FUNCTION_BLOCK FB_System_HES_991
VAR_INPUT
	Freigabe_auto				: BOOL;
	Freigabe_Deakt_auto			: BOOL;
	Betrieb_Anford_auto			: BOOL;

END_VAR
VAR_OUTPUT
	{attribute 'OPC.UA.DA' := '1'}Steuerung				: ST_System_HES_Steuerung;		
	{attribute 'OPC.UA.DA' := '1'}Stellwert				: ST_System_HES_Stellwert;		
	{attribute 'OPC.UA.DA' := '1'}Zustand					: ST_System_HES_Zustand;	
	{attribute 'OPC.UA.DA' := '1'}Parameter				: ST_System_HES_Parameter;		
END_VAR
VAR
	Pumpe_191					: FB_PU_191;
	Stellventil_191				: FB_SV;
	HybriderEnergiespeicher_991	: FB_HES;

	Zustandscheck			: FB_System_HES_Zustandscheck;
	Logik					: FB_System_HES_Logik;
	Ablaufsteuerung			: FB_System_HES_Ablaufsteuerung;
	Ablaufsteuerung_191		: FB_System_HES_Ablaufsteuerung;

END_VAR
VAR // added by the converter: edge detectors and wires of the graphical bodies
    _w1, _w4, _w6 : ANY;
    _w2, _w3, _w5 : BOOL;
END_VAR

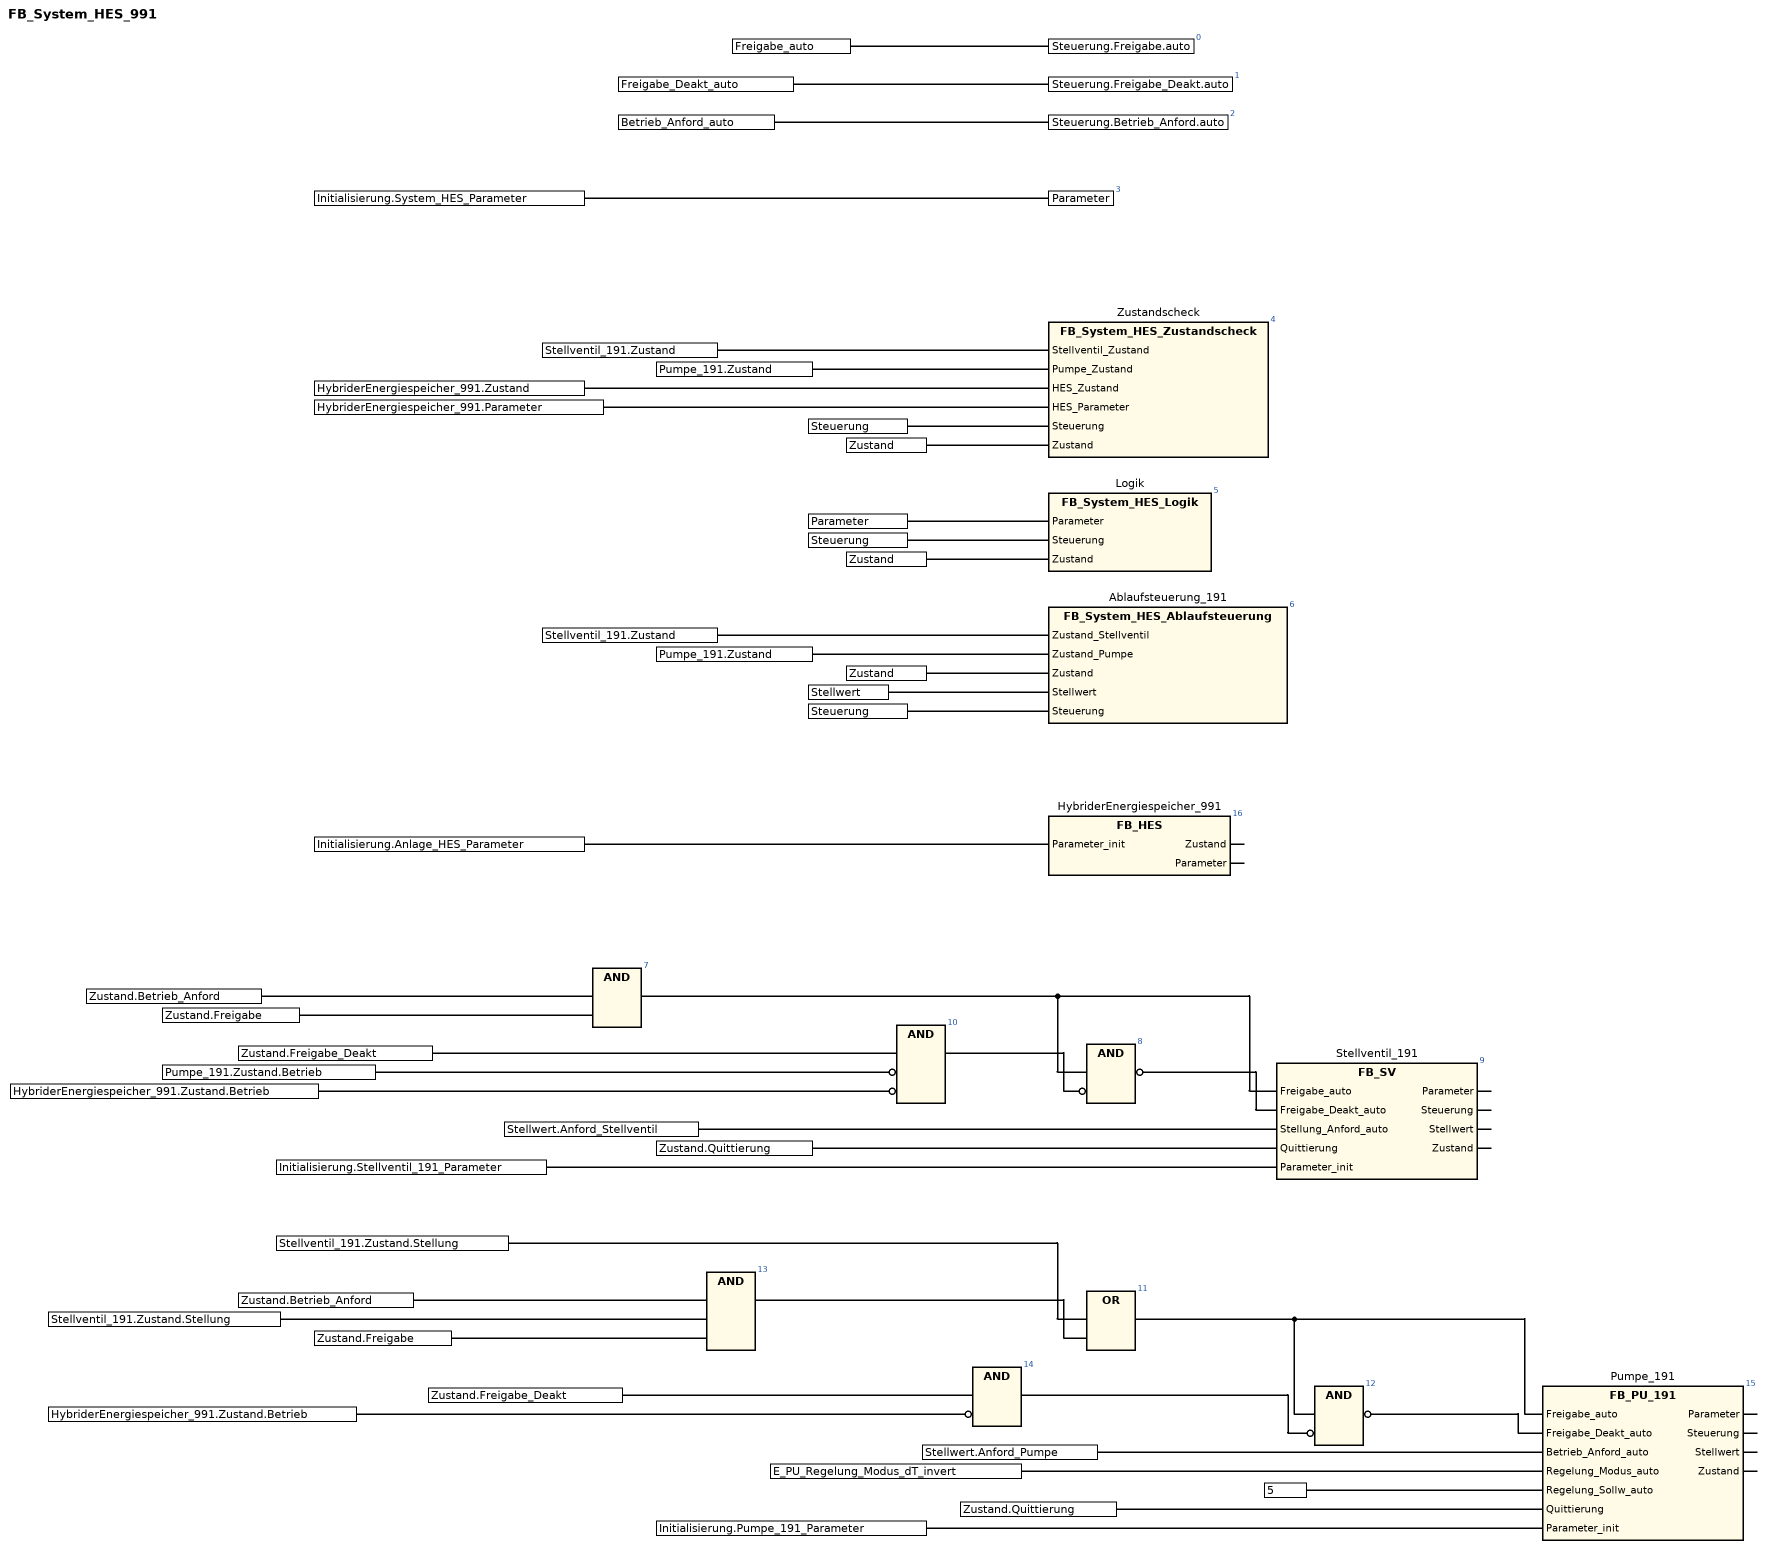
Steuerung.Freigabe.auto := Freigabe_auto;
Steuerung.Freigabe_Deakt.auto := Freigabe_Deakt_auto;
Steuerung.Betrieb_Anford.auto := Betrieb_Anford_auto;
Parameter := Initialisierung.System_HES_Parameter;
Zustandscheck(
    Stellventil_Zustand := Stellventil_191.Zustand,
    Pumpe_Zustand := Pumpe_191.Zustand,
    HES_Zustand := HybriderEnergiespeicher_991.Zustand,
    HES_Parameter := HybriderEnergiespeicher_991.Parameter,
    Steuerung := Steuerung,
    Zustand := Zustand); // FB_System_HES_Zustandscheck
Logik(Parameter := Parameter, Steuerung := Steuerung, Zustand := Zustand); // FB_System_HES_Logik
Ablaufsteuerung_191(
    Zustand_Stellventil := Stellventil_191.Zustand,
    Zustand_Pumpe := Pumpe_191.Zustand,
    Zustand := Zustand,
    Stellwert := Stellwert,
    Steuerung := Steuerung); // FB_System_HES_Ablaufsteuerung
_w1 := Zustand.Betrieb_Anford AND Zustand.Freigabe;
Stellventil_191(
    Freigabe_auto := _w1,
    Freigabe_Deakt_auto := NOT (_w1 AND NOT _w2),
    Stellung_Anford_auto := Stellwert.Anford_Stellventil,
    Quittierung := Zustand.Quittierung,
    Parameter_init := Initialisierung.Stellventil_191_Parameter); // FB_SV
_w2 := Zustand.Freigabe_Deakt AND NOT Pumpe_191.Zustand.Betrieb AND NOT HybriderEnergiespeicher_991.Zustand.Betrieb;
_w4 := Stellventil_191.Zustand.Stellung OR _w3;
_w6 := _w4 AND NOT _w5;
_w3 := Zustand.Betrieb_Anford AND Stellventil_191.Zustand.Stellung AND Zustand.Freigabe;
_w5 := Zustand.Freigabe_Deakt AND NOT HybriderEnergiespeicher_991.Zustand.Betrieb;
Pumpe_191(
    Freigabe_auto := _w4,
    Freigabe_Deakt_auto := NOT _w6,
    Betrieb_Anford_auto := Stellwert.Anford_Pumpe,
    Regelung_Modus_auto := E_PU_Regelung_Modus_dT_invert,
    Regelung_Sollw_auto := 5,
    Quittierung := Zustand.Quittierung,
    Parameter_init := Initialisierung.Pumpe_191_Parameter); // FB_PU_191
HybriderEnergiespeicher_991(Parameter_init := Initialisierung.Anlage_HES_Parameter); // FB_HES

END_FUNCTION_BLOCK

(* stored: Version 1.1.0.1, ProductVersion 3.1.4024.9
   POU FB_System_HES_991: Id {dfb2cec3-2b14-4ed7-b8ad-4454b8cf9bdd}, SpecialFunc None *)
